FUNCTION_BLOCK FB_BaseTelescopeControl
VAR_INPUT
	bInit				: BOOL;
	bPark				: BOOL;
	bSlew				: BOOL;
	bTrack				: BOOL;
	bStop				: BOOL;
	
	bBrakeClearing		: BOOL	:= TRUE;
	
	telescopeConfig		: ST_TelescopeConfig;
END_VAR
VAR_OUTPUT
	bPower				: BOOL;
	bError				: BOOL;
	bReset				: BOOL;
END_VAR
VAR
	comm				: I_Comm;
	
	fbMachine			: FB_TelescopeMachine;
	fbParkedState		: FB_TelescopeParkedState(fbMachine);
	fbInitializingState	: FB_TelescopeInitializingState(fbMachine);
	fbParkingState		: FB_TelescopeParkingState(fbMachine);
	fbIdleState			: FB_TelescopeIdleState(fbMachine);
	fbSlewingState		: FB_TelescopeSlewingState(fbMachine);
	fbTrackingState		: FB_TelescopeTrackingState(fbMachine);
	
	bPowerFailure		: BOOL;		// triggers power-failure event
	
	fbTime				: FB_AstroClock;	// precise astronomical	time
	fJD					: LREAL;	// current Julian Date calculated from system time
	fLST				: LREAL;	// local siderial time calculated from Julian date

	TCSpowerEvent,
	TCSgohomeEvent,
	TCSparkEvent,
	TCSgotoEvent,
	TCStrackEvent,
	TCSstopEvent,
	AltitudeEvent,
	TCSreadyEvent,
	TCSCTOEvent			: FB_Eventlog;
END_VAR

// get the system time
fbTime();
fJD := DateTime2JD(fbTime.time_RTCEX2);
fLST := CT2LST(telescopeConfig.longitude, fJD);

// run the state machine
fbMachine(
	bInit				:= bInit,
	bPark				:= bPark,
	bSlew 				:= bSlew,
	bTrack 				:= bTrack,
	bStop 				:= bStop,
	fbParkedState		:= fbParkedState,
	fbInitializingState	:= fbInitializingState,
	fbParkingState		:= fbParkingState,
	fbIdleState			:= fbIdleState,
	fbSlewingState		:= fbSlewingState,
	fbTrackingState		:= fbTrackingState,	
);

bInit	:= FALSE;
bPark	:= FALSE;
bSlew 	:= FALSE;
bTrack 	:= FALSE;
bStop 	:= FALSE;

METHOD _Initialize : BOOL
VAR_INPUT
END_VAR
END_METHOD

METHOD _Park : BOOL
VAR_INPUT
END_VAR
END_METHOD

METHOD FB_init : BOOL
VAR_INPUT
	bInitRetains : BOOL; // if TRUE, the retain variables are initialized (warm start / cold start)
	bInCopyCode : BOOL;  // if TRUE, the instance afterwards gets moved into the copy code (online change)
	comm			: I_Comm;	
END_VAR
THIS^.comm := comm;
END_METHOD

END_FUNCTION_BLOCK

(* stored: Version 1.1.0.1, ProductVersion 3.1.4024.15
   POU FB_BaseTelescopeControl: Id {eddbf876-a986-4fe1-ba5b-16d782882b92}, SpecialFunc None
   Method _Initialize: Id {f5caea65-cedf-4c3b-8428-6180ca9de8c7}
   Method _Park: Id {f5cfd253-b848-4530-8152-490bf96244a1}
   Method FB_init: Id {a32d2f32-4a31-4d05-8712-e937ed61ba13} *)
